(* CoDeSys 2.3.9.59 project: PD2.pro *)
(* Libraries: Standard.lib, SYSLIBCALLBACK.LIB *)

(* PLC configuration (modules and I/O channels)
Configuration EC4P-200 [Root] node -1, in %IB0 out %QB0 {EC4P_RestartPwrOn = WARMSTART; EC4P_MaxCycleTime = 20; EC4P_Com1BaudRate = 38400; EC4P_CAN1BaudRate = 125KBaud; EC4P_RoutingId = 127; EC4P_EasyNetId = 1; EC4P_EasyNetCfg = 0; EC4P_EasyNetCycleTime = 50; EC4P_RoutingChannel = CAN1; EC4P_IPFlags = 0; EC4P_IPAddress = 0; EC4P_SubNetMask = 0; EC4P_DefaultGateway = 0; EC4P_SummerWinterFlags = 0; EC4P_SummerWinterRule1 = 0; EC4P_SummerWinterRule2 = 0}
  Local I/O [EC4P_LocalIO] node 0, in %IB0 out %QB0 {EC4P_LocalInt = 0}
    I1 AT %IX0.0 [LocalBitInput] Input I1
    I2 AT %IX0.1 [LocalBitInput] Input I2
    I3 AT %IX0.2 [LocalBitInput] Input I3
    I4 AT %IX0.3 [LocalBitInput] Input I4
    I5 AT %IX0.4 [LocalBitInput] Input I5
    I6 AT %IX0.5 [LocalBitInput] Input I6
    I7 AT %IX0.6 [LocalBitInput] Input I7
    I8 AT %IX0.7 [LocalBitInput] Input I8
    I9 AT %IX1.0 [LocalBitInput] Input I9
    I10 AT %IX1.1 [LocalBitInput] Input I10
    I11 AT %IX1.2 [LocalBitInput] Input I11
    I12 AT %IX1.3 [LocalBitInput] Input I12
    I13 AT %IX1.4 [LocalDiagInput] Diagnostic Input I13
    I14 AT %IX1.5 [LocalDiagInput] Diagnostic Input I14
    I15 AT %IX1.6 [LocalDiagInput] Diagnostic Input I15
    I16 AT %IX1.7 [LocalDiagInput] Diagnostic Input I16
    I7_Analog AT %IW2 [LocalAnalogIn] Input I7, 10Bit, 0-10VDC
    I8_Analog AT %IW4 [LocalAnalogIn] Input I8, 10Bit, 0-10VDC
    I11_Analog AT %IW6 [LocalAnalogIn] Input I11, 10Bit, 0-10VDC
    I12_Analog AT %IW8 [LocalAnalogIn] Input I12, 10Bit, 0-10VDC
    Transistor Outputs [EC4P_TOutputs] node 0, in %IB10 out %QB0
      Q1 AT %QX0.0 [LocalBitOutput] Transistor-Output Q1
      Q2 AT %QX0.1 [LocalBitOutput] Transistor-Output Q2
      Q3 AT %QX0.2 [LocalBitOutput] Transistor-Output Q3
      Q4 AT %QX0.3 [LocalBitOutput] Transistor-Output Q4
      Q5 AT %QX0.4 [LocalBitOutput] Transistor-Output Q5
      Q6 AT %QX0.5 [LocalBitOutput] Transistor-Output Q6
      Q7 AT %QX0.6 [LocalBitOutput] Transistor-Output Q7
      Q8 AT %QX0.7 [LocalBitOutput] Transistor-Output Q8
    No Analog Output [EC4P_NoAnalogOutput] node 1, in %IB10 out %QB1
    No Keys [EC4P_NoKeys] node 2, in %IB10 out %QB1
    No Counter [EC4P_NoCounter] node 3, in %IB10 out %QB1
  Extension [EC4P_Extension] node 1, in %IB10 out %QB1
    No Extension [EC4P_NoExtension] node 0, in %IB10 out %QB1
*)

(* POU PLC_PRG, LD *)
PROGRAM PLC_PRG
VAR
END_VAR
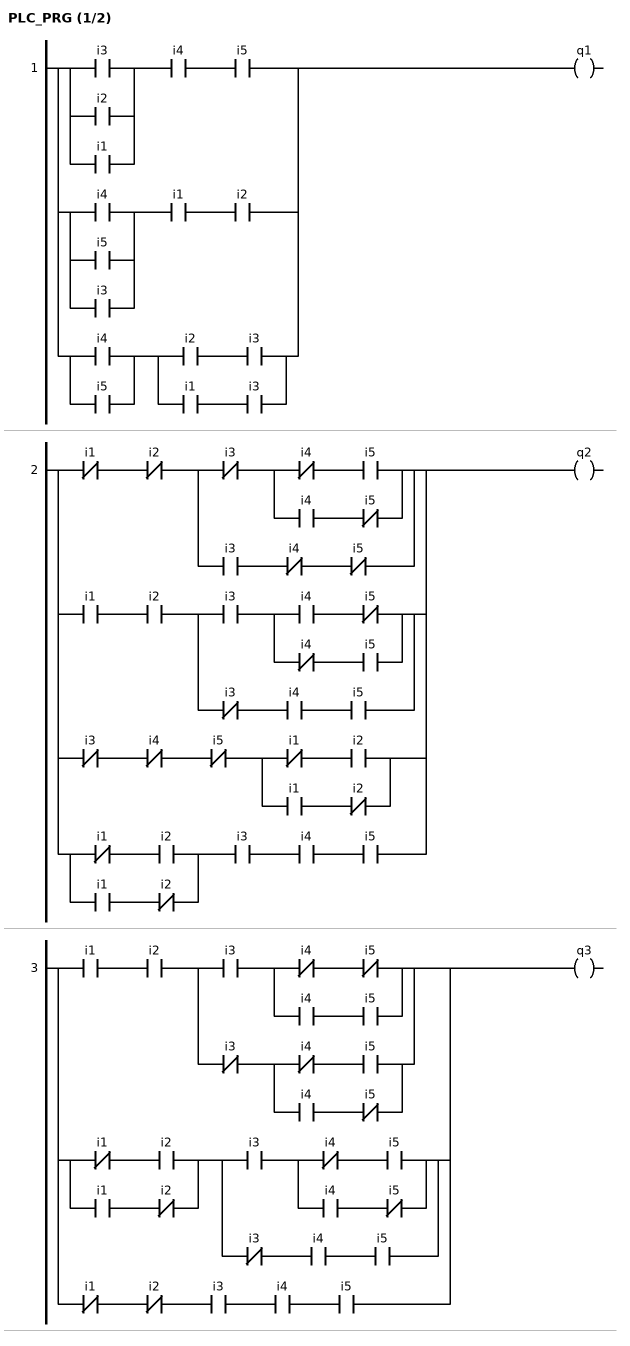
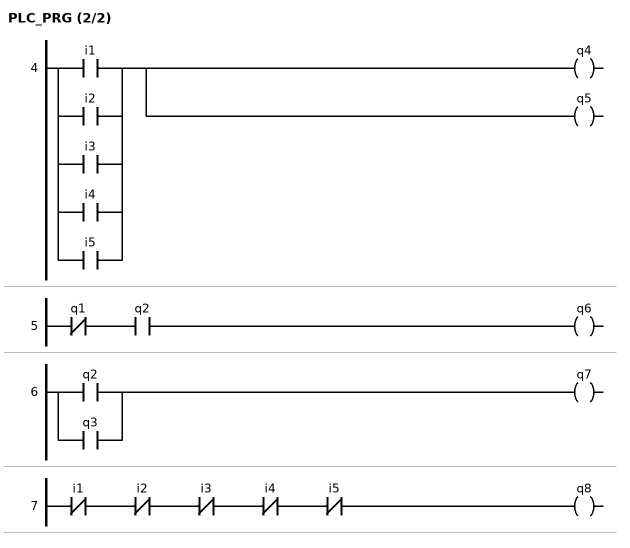
_LD_ (* Ladder Diagram *)
NETWORK 1
	{ { [i3] | [i2] | [i1] } - [i4] - [i5] | { [i4] | [i5] | [i3] } - [i1] - [i2] | { [i4] | [i5] } - { [i2] - [i3] | [i1] - [i3] } } --- (q1)
NETWORK 2
	{ [/i1] - [/i2] - { [/i3] - { [/i4] - [i5] | [i4] - [/i5] } | [i3] - [/i4] - [/i5] } | [i1] - [i2] - { [i3] - { [i4] - [/i5] | [/i4] - [i5] } | [/i3] - [i4] - [i5] } | [/i3] - [/i4] - [/i5] - { [/i1] - [i2] | [i1] - [/i2] } | { [/i1] - [i2] | [i1] - [/i2] } - [i3] - [i4] - [i5] } --- (q2)
NETWORK 3
	{ [i1] - [i2] - { [i3] - { [/i4] - [/i5] | [i4] - [i5] } | [/i3] - { [/i4] - [i5] | [i4] - [/i5] } } | { [/i1] - [i2] | [i1] - [/i2] } - { [i3] - { [/i4] - [i5] | [i4] - [/i5] } | [/i3] - [i4] - [i5] } | [/i1] - [/i2] - [i3] - [i4] - [i5] } --- (q3)
NETWORK 4
	{ [i1] | [i2] | [i3] | [i4] | [i5] } --- (q4) (q5)
NETWORK 5
	[/q1] - [q2] --- (q6)
NETWORK 6
	{ [q2] | [q3] } --- (q7)
NETWORK 7
	[/i1] - [/i2] - [/i3] - [/i4] - [/i5] --- (q8)
_END_LD_
(* the same logic as Structured Text *)
(* Network 1 *)
q1 := (i3 OR i2 OR i1) AND i4 AND i5 OR (i4 OR i5 OR i3) AND i1 AND i2 OR (i4 OR i5) AND (i2 AND i3 OR i1 AND i3);
(* Network 2 *)
q2 := NOT i1 AND NOT i2 AND (NOT i3 AND (NOT i4 AND i5 OR i4 AND NOT i5) OR i3 AND NOT i4 AND NOT i5) OR i1 AND i2 AND (i3 AND (i4 AND NOT i5 OR NOT i4 AND i5) OR NOT i3 AND i4 AND i5) OR NOT i3 AND NOT i4 AND NOT i5 AND (NOT i1 AND i2 OR i1 AND NOT i2) OR (NOT i1 AND i2 OR i1 AND NOT i2) AND i3 AND i4 AND i5;
(* Network 3 *)
q3 := i1 AND i2 AND (i3 AND (NOT i4 AND NOT i5 OR i4 AND i5) OR NOT i3 AND (NOT i4 AND i5 OR i4 AND NOT i5)) OR (NOT i1 AND i2 OR i1 AND NOT i2) AND (i3 AND (NOT i4 AND i5 OR i4 AND NOT i5) OR NOT i3 AND i4 AND i5) OR NOT i1 AND NOT i2 AND i3 AND i4 AND i5;
(* Network 4 *)
q4 := i1 OR i2 OR i3 OR i4 OR i5;
q5 := q4;
(* Network 5 *)
q6 := NOT q1 AND q2;
(* Network 6 *)
q7 := q2 OR q3;
(* Network 7 *)
q8 := NOT i1 AND NOT i2 AND NOT i3 AND NOT i4 AND NOT i5;
END_PROGRAM

(* Visualisation seg_7
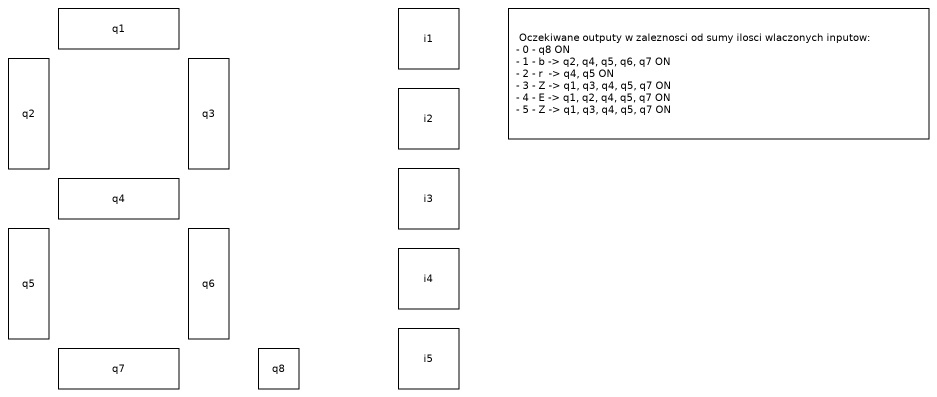
rectangle at (130,30)-(251,71): text "q1"; alarm colour if q1; toggles q1
rectangle at (260,80)-(301,191): text "q3"; alarm colour if q3; toggles q3
rectangle at (80,80)-(121,191): text "q2"; alarm colour if q2; toggles q2
rectangle at (130,200)-(251,241): text "q4"; alarm colour if q4; toggles q4
rectangle at (260,250)-(301,361): text "q6"; alarm colour if q6; toggles q6
rectangle at (80,250)-(121,361): text "q5"; alarm colour if q5; toggles q5
rectangle at (130,370)-(251,411): text "q7"; alarm colour if q7; toggles q7
rectangle at (330,370)-(371,411): text "q8"; alarm colour if q8; toggles q8
rectangle at (470,30)-(531,91): text "i1"; alarm colour if i1; toggles i1
rectangle at (470,110)-(531,171): text "i2"; alarm colour if i2; toggles i2
rectangle at (470,190)-(531,251): text "i3"; alarm colour if i3; toggles i3
rectangle at (470,350)-(531,411): text "i5"; alarm colour if i5; toggles i5
rectangle at (470,270)-(531,331): text "i4"; alarm colour if i4; toggles i4
rectangle at (580,30)-(1001,161): text "Oczekiwane outputy w zaleznosci od sumy ilosci wlaczonych inputow: / - 0 - q8 ON / - 1 - b -> q2, q4, q5, q6, q7 ON / - 2 - r  -> q4, q5 ON / - 3 - Z -> q1, q3, q4, q5, q7 ON / - 4 - E -> q1, q2, q4, q5, q7 ON / - 5 - Z -> q1, q3, q4, q5, q7 ON"
*)
